// TwinCAT 3 PLC project plc
// ProgramVersion: 3.1.4024.0
// libraries:
//   Tc2_Standard, * (Beckhoff Automation GmbH)
//   Tc2_System, * (Beckhoff Automation GmbH)
//   Tc3_Module, * (Beckhoff Automation GmbH)
// project tree:
//   DUTs/ Axis_output.TcDUT, Axis_STATUS.TcDUT
//   / PlcTask.TcTTO
//   POUs/ MAIN.TcPOU
// real-time tasks:
//   TASK PlcTask: cycle T#1ms, priority 4, ADS port 350
// I/O:
//   DEVICE Device 2 (EtherCAT), AmsNetId 169.254.115.184.3.1
//     Drive 3 (MBDLN25BE) [MBDLN25BE]
//     Drive 4 (MBDLN25BE) [MBDLN25BE] (disabled)
//     Box 5 (EV1616DN) [SCATECH EV1616DN] (disabled)
// variable links:
//   plc/plc Instance <-> Device 2 (EtherCAT)/Box 5 (EV1616DN)
//     PlcTask Outputs/MAIN.BREAK0 <-> OUTPUT BITS process data mapping/OUT1
//     PlcTask Outputs/MAIN.BREAK1 <-> OUTPUT BITS process data mapping/OUT2
//   plc/plc Instance <-> Device 2 (EtherCAT)/Drive 3 (MBDLN25BE)
//     PlcTask Inputs/MAIN.Axis0_status/Actual_Position <-> Transmit PDO mapping 1/Position actual value
//     PlcTask Inputs/MAIN.Axis0_status/Actual_Torque <-> Transmit PDO mapping 1/Torque actual value
//     PlcTask Inputs/MAIN.Axis0_status/Actual_Velocity <-> Transmit PDO mapping 1/Velocity actual value
//     PlcTask Inputs/MAIN.Axis0_status/Following_error <-> Transmit PDO mapping 1/Following error actual value
//     PlcTask Inputs/MAIN.Axis0_status/Mode_of_Operation_disp <-> Transmit PDO mapping 1/Modes of operation display
//     PlcTask Inputs/MAIN.Axis0_status/Status <-> Transmit PDO mapping 1/Statusword
//     PlcTask Outputs/MAIN.Axis0/Control_Word <-> Receive PDO mapping 1/Controlword
//     PlcTask Outputs/MAIN.Axis0/Max_Velocity <-> Receive PDO mapping 1/Max motor speed
//     PlcTask Outputs/MAIN.Axis0/Mode_of_Operation <-> Receive PDO mapping 1/Modes of operation
//     PlcTask Outputs/MAIN.Axis0/Profile_Velocity <-> Receive PDO mapping 1/Profile velocity
//     PlcTask Outputs/MAIN.Axis0/Target_Position <-> Receive PDO mapping 1/Target position
//   plc/plc Instance <-> Device 2 (EtherCAT)/Drive 4 (MBDLN25BE)
//     PlcTask Inputs/MAIN.Axis1_status/Actual_Position <-> Transmit PDO mapping 1/Position actual value
//     PlcTask Inputs/MAIN.Axis1_status/Actual_Torque <-> Transmit PDO mapping 1/Torque actual value
//     PlcTask Inputs/MAIN.Axis1_status/Actual_Velocity <-> Transmit PDO mapping 1/Velocity actual value
//     PlcTask Inputs/MAIN.Axis1_status/Following_error <-> Transmit PDO mapping 1/Following error actual value
//     PlcTask Inputs/MAIN.Axis1_status/Mode_of_Operation_disp <-> Transmit PDO mapping 1/Modes of operation display
//     PlcTask Inputs/MAIN.Axis1_status/Status <-> Transmit PDO mapping 1/Statusword
//     PlcTask Outputs/MAIN.Axis1/Control_Word <-> Receive PDO mapping 1/Controlword
//     PlcTask Outputs/MAIN.Axis1/Max_Velocity <-> Receive PDO mapping 1/Max motor speed
//     PlcTask Outputs/MAIN.Axis1/Mode_of_Operation <-> Receive PDO mapping 1/Modes of operation
//     PlcTask Outputs/MAIN.Axis1/Profile_Velocity <-> Receive PDO mapping 1/Profile velocity
//     PlcTask Outputs/MAIN.Axis1/Target_Position <-> Receive PDO mapping 1/Target position

CONFIGURATION plc
    RESOURCE PLC ON TwinCAT3
        TASK PlcTask(INTERVAL := T#1ms, PRIORITY := 4);
        PROGRAM MAIN WITH PlcTask : MAIN;
    END_RESOURCE
END_CONFIGURATION

// ---- DUTs/Axis_output.TcDUT
TYPE Axis_output :
STRUCT
	Control_Word AT%Q*:WORD;
	Target_Position AT%Q*:DINT;
	Profile_Velocity AT%Q*:UDINT;
	Max_Velocity AT%Q*:UDINT;
	Mode_of_Operation AT%Q* :BYTE:=1;
END_STRUCT
END_TYPE

// ---- DUTs/Axis_STATUS.TcDUT
TYPE Axis_STATUS :
STRUCT
	Status : WORD;
	Mode_of_Operation_disp:BYTE;
	Actual_Position:DINT;
	Actual_Velocity :DINT;
	Following_error:DINT;
	Actual_Torque:INT;
END_STRUCT
END_TYPE

// ---- POUs/MAIN.TcPOU
PROGRAM MAIN
VAR
	Axis0 AT%QD0:Axis_output;
	Axis1 AT%QD5:Axis_output;
	Axis0_status AT%ID0:Axis_STATUS;
	Axis1_status AT%ID5:Axis_STATUS;
	BREAK0 AT%QD100 :BOOL:=0;
	BREAK1 AT%QD101 :BOOL:=0;
END_VAR

END_PROGRAM
